// NETWORK 3
// label: //'SEPARATE2 COLET'
fbPiston[9](
    stPISTON := stPISTON_PARAM[9],
    bDepened_open1 := TRUE,
    bDepened_open2 := TRUE,
    bDepened_close1 := TRUE,
    bDepened_close2 := TRUE); // FB_PISTON

// NETWORK 4
// label: //'SEPARATE2 PULL'
fbPiston[10](
    stPISTON := stPISTON_PARAM[10],
    bDepened_open1 := TRUE,
    bDepened_open2 := TRUE,
    bDepened_close1 := TRUE,
    bDepened_close2 := TRUE); // FB_PISTON

// NETWORK 5
// label: //'SEPARATE2 TRAY'
fbPiston[11](
    stPISTON := stPISTON_PARAM[11],
    bDepened_open1 := TRUE,
    bDepened_open2 := TRUE,
    bDepened_close1 := TRUE,
    bDepened_close2 := TRUE); // FB_PISTON

// NETWORK 6
// label: //'SEPARATE2 PUSH PINS'
fbPiston[12](
    stPISTON := stPISTON_PARAM[7],
    bDepened_open1 := TRUE,
    bDepened_open2 := TRUE,
    bDepened_close1 := TRUE,
    bDepened_close2 := TRUE); // FB_PISTON

// NETWORK 7
// label: //'SEPARATE2 TRAY PUSHER'
fbPiston[18](
    stPISTON := stPISTON_PARAM[18],
    bDepened_open1 := TRUE,
    bDepened_open2 := TRUE,
    bDepened_close1 := TRUE,
    bDepened_close2 := TRUE); // FB_PISTON

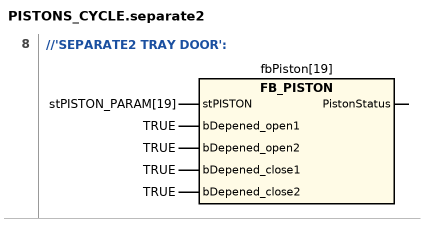
// NETWORK 8
// label: //'SEPARATE2 TRAY DOOR'
fbPiston[19](
    stPISTON := stPISTON_PARAM[19],
    bDepened_open1 := TRUE,
    bDepened_open2 := TRUE,
    bDepened_close1 := TRUE,
    bDepened_close2 := TRUE); // FB_PISTON
END_ACTION

END_PROGRAM

// ---- GlobalTextList.TcGTLO
TEXTLIST GlobalTextList
  491 = '#%d'
  711 = '+'
  478 = '-'
  1486 = '?'
  1979 = 'Axis Error'
  943 = 'axis: %s'
  779 = 'Continous'
  1966 = 'Drive Err: %x'
  206 = 'Enabled'
  743 = 'Fast'
  1321 = 'home'
  928 = 'Home Done'
  799 = 'Home mode Direct'
  1171 = 'Home sensor'
  860 = 'Inching'
  18 = 'Limited Operation(E-Stop)'
  610 = 'MC Err: %x'
  10 = 'MC Error'
  417 = 'Mod Pos: %.1f [deg]'
  252 = 'Modulo'
  1438 = 'Modulo Position'
  1253 = 'Pos: %.1f [units]'
  82 = 'Power'
  466 = 'Power Off'
  1360 = 'Power On - Home Done'
  1642 = 'Power On - Not Homed'
  633 = 'reset'
  553 = 'Slow'
  54 = 'step size: %.1f [units/sec]'
  430 = 'stop'
  324 = 'Vel: %.1f [units/s]'
  237 = 'velocity: %.1f [units/sec]'
END_TEXTLIST
